PROGRAM MAIN
VAR
END_VAR

END_PROGRAM

(* stored: Version 1.1.0.1
   POU MAIN: Id {f886aa28-2104-4b1d-9bce-b8a04f8fd61c} *)
